# EPICS autosave request: iocBoot/gmca_23b_ioc2/dbSave/BD_Dh_.req
%
% BURT Request File
%
% $(P)BD:Dh: Horizontal Beam Delivery (type: Downstream Support)
%

file assy.req ASSY=$(P)BD:Dh
$(P)BD:Dh:BaseLength
$(P)BD:Dh:RotOrigin
file mtr1.req MTR1=$(P)BD:mhd
file mtr1.req MTR1=$(P)BD:mhu
file drv1.req DRV1=$(P)BD:HDS
file drv1.req DRV1=$(P)BD:HUS
file axs1.req AXS1=$(P)BD:HD
file axs1.req AXS1=$(P)BD:HA
